FUNCTION_BLOCK FB_CoreSwaging
VAR_INPUT
END_VAR
VAR_OUTPUT
END_VAR
VAR
    iState : INT := 0;
	FeedbackTimer : TON;
    DelayTimer : TON;
	fSetAlarm : FB_SetAlarm;
	fCheckFeedback : FB_CheckFeedback;
END_VAR

CASE iState OF
	0: (* Idle/Off, DI_ECS=FALSE *)
		(* Manual Mode Handling *)
		IF GVL_HMI.i_nCoreSwagingMode = 1 THEN
			IF GVL_IO.DI_JLU THEN (* Jog switch pressed *)
				(* Motor M3 runs infinitely while switch is pressed *)
				iState := 10;
			END_IF
		ELSE
			iState := 10;
		END_IF
		
	10: (* check safety conditions *)
		IF GVL_HMI.bSafeties AND GVL_IO.DI_ECS THEN (* Safeties OK and Enable Switch On *)
            GVL_IO.DO_M1 := TRUE; (* Start Oil Pump *)
			CheckFeedback(E_FT.PUMP);
			IF GVL_IO.DI_M1 THEN
				DelayAndAdvance(GVL_InitialSetting.PUMP_RunningDelayTime, iState+10);
			END_IF
        END_IF
		
    20: (* Ensure CYL6 is Extended *)
        IF NOT GVL_IO.DI_CYL6_E THEN
			GVL_IO.DO_SV1 := TRUE;	// Power Pack Hydraulic Pressure Relief Valve
            GVL_IO.DO_CYL6_E := TRUE;
			CheckFeedback(E_FT.CYL6_E);
        ELSE
			DelayAndAdvance(GVL_InitialSetting.CYLINDER6EXTENDED_RunningDelayTime, iState+1);
        END_IF
	21: (* Ensure CYL5 is Retracted *)
    	IF NOT GVL_IO.DI_CYL5_R THEN
			GVL_IO.DO_CYL5_R := TRUE;
			CheckFeedback(E_FT.CYL5_R);
		ELSE
			iState := (iState + 10) / 10 * 10;
		END_IF
		
    30: (* Ensure CYL7 is Retracted *)
        IF NOT GVL_IO.DI_CYL7_R THEN
            GVL_IO.DO_CYL7_R := TRUE;
			CheckFeedback(E_FT.CYL7_R);
        ELSE
			DelayAndAdvance(GVL_InitialSetting.CYLINDER7RETRACTED_RunningDelayTime, iState+10);
        END_IF
    
    40: (* Low Lead Spool Check *)
        IF NOT GVL_IO.DI_PE5 THEN
			fSetAlarm( sMsg := GVL_AlarmMessage.PE5_FAIL );
        ELSE
			IF GVL_IO.DI_CYL4_R THEN
				(* index M3 *)
				
				iState := iState + 1;
			END_IF
        END_IF
	41: 
		DelayAndAdvance(GVL_InitialSetting.M3_RunningDelayTime, (iState + 10) / 10 * 10);
    
    50: (* Extend CYL7 *)
        IF NOT GVL_IO.DI_CYL7_E THEN
			GVL_IO.DO_CYL7_E := TRUE;
			CheckFeedback(E_FT.CYL7_E);
        ELSE
			DelayAndAdvance(GVL_InitialSetting.CYLINDER7EXTENDED_RunningDelayTime, iState + 10);
        END_IF
    
    60: (* Retract CYL6 *)
        IF NOT GVL_IO.DI_CYL6_R THEN
			GVL_IO.DO_CYL6_R := TRUE;
			CheckFeedback(E_FT.CYL6_R);
        ELSE
			DelayAndAdvance(GVL_InitialSetting.CYLINDER6RETRACTED_RunningDelayTime, iState + 10);
        END_IF
    
    70: (* Extend CYL5 *)
        IF NOT GVL_IO.DI_CYL5_E THEN
			GVL_IO.DO_CYL5_E := TRUE;
			CheckFeedback(E_FT.CYL5_E);
        ELSE
			DelayAndAdvance(GVL_InitialSetting.CYLINDER5EXTENDED_RunningDelayTime, iState + 10);
        END_IF
    
    80: (* Retract CYL5 *)
        IF NOT GVL_IO.DI_CYL5_R THEN
			GVL_IO.DO_CYL5_R := TRUE;
			CheckFeedback(E_FT.CYL5_R);
		ELSE
			DelayAndAdvance(GVL_InitialSetting.CYLINDER5RETRACTED_RunningDelayTime, iState + 10);
        END_IF
		
	90: (* Future Step *)
		iState := 20;
END_CASE

METHOD CheckFeedback : BOOL
VAR_INPUT
	t : E_FT;
END_VAR
VAR_OUTPUT
	o_nResult : INT := 0;	// -1: fail, 0: checking, 1: success 
END_VAR
fCheckFeedback(t:=t, FeedbackTimer:=FeedbackTimer);
o_nResult := fCheckFeedback.o_nResult;
END_METHOD

METHOD DelayAndAdvance : BOOL
VAR_INPUT
	i_nDelayTime: INT;	// ms
	i_nNextState: INT;
END_VAR

VAR
END_VAR
IF NOT DelayTimer.IN THEN
    DelayTimer(IN := TRUE, PT := INT_TO_TIME(i_nDelayTime));
ELSE
    IF DelayTimer.Q THEN 
        iState := i_nNextState; 
    END_IF
END_IF
END_METHOD

END_FUNCTION_BLOCK

(* stored: Version 1.1.0.1, ProductVersion 3.1.4024.6
   POU FB_CoreSwaging: Id {32bb99d5-55a6-44d7-8d53-4198850662e4}, SpecialFunc None
   Method CheckFeedback: Id {ca45cbb6-be73-4478-acca-2fc864d4bbed}
   Method DelayAndAdvance: Id {532274d9-37b2-4f3d-a542-0cdcb8beabdd} *)
